// TIA Portal V17 export
// export: Created 2024-08-29T18:23:50.8761103Z, ExportSetting WithDefaults, DisplayName Totally Integrated Automation Portal, DisplayVersion V17 Update 7, DisplayName TIA Portal Openness, DisplayVersion V17 Update 7, DisplayName TIA Portal Version Control Interface, DisplayVersion V17, DisplayName SINAMICS Startdrive Advanced, DisplayVersion V17 SP2, DisplayName SINAMICS Startdrive G110M, G120, G120C, G120D, G120P, G115D, DisplayVersion V17 SP2, DisplayName SINAMICS Startdrive G130, G150, S120, S150, SINAMICS MV, S210, DisplayVersion V17 SP2, DisplayName STEP 7 Professional, DisplayVersion V17 Update 7, DisplayName STEP 7 Safety, DisplayVersion V17 Update 6, DisplayName WinCC Advanced / Unified PC, DisplayVersion V17 Update 7
VAR_GLOBAL   // PLC tag table "programMemory"
   cycleTimeReset AT %M250.1 : Bool;
   clearData AT %M250.0 : Bool;
   programAutoModeSelection AT %M250.3 : Bool;
   productInNest AT %M250.2 : Bool;
   bypass1 AT %M2.0 : Bool;
   bypass2 AT %M2.1 : Bool;
   bypass3 AT %M2.2 : Bool;
END_VAR
